(* Logix 5000 project; controller Safety vendor 1 type 14 code 86 rev 19.11; software revision 19.01; part 6 of 17 *)
(* tags used below, declared in another part *)
   ChgMe : BOOL;
   ESTOP_x201PB040 : DCI_STOP;   // OS1 Line EStop Pushbutton
   ESTOP_x211PB040 : DCI_STOP;   // OS2 Line EStop Pushbutton
   ESTOP_x221PB040 : DCI_STOP;   // OS3 Line EStop Pushbutton
   ESTOP_x231PB040 : DCI_STOP;   // OS4N Line EStop Pushbutton
   ESTOP_x241PB040 : DCI_STOP;   // OS4S Line EStop Pushbutton
   ESTOP_x251PB040 : DCI_STOP;   // OS5 Line EStop Pushbutton
   ESTOP_x261PB040 : DCI_STOP;   // OS6 Line EStop Pushbutton
   ESTOP_x271PB040 : DCI_STOP;   // OS8 Line EStop Pushbutton
   ESTOP_x281PB040 : DCI_STOP;   // OS9 Line EStop Pushbutton
   ESTOP_x291PB040 : DCI_STOP;   // OS11 Line EStop Pushbutton
   ESTOP_x301PB040 : DCI_STOP;   // OS13 Line EStop Pushbutton
   ESTOP_x311PB040 : DCI_STOP;   // OS14 Line EStop Pushbutton
   ESTOP_x311PB130 : DCI_STOP;   // OS14 Shear Estop Pushbutton
   ESTOP_x321PB040 : DCI_STOP;   // OS15 Line EStop Pushbutton
   ESTOP_x331PB040 : DCI_STOP;   // OS16 Line EStop Pushbutton
   ESTOP_x480PB470 : DCI_STOP;   // DPD Line EStop Pushbutton
   ESTOP_x480PB550 : DCI_STOP;   // DPD (In Pit) Line EStop Pushbutton
   ESTOP_x519LS470 : DCI_STOP;   // G1 Tripwire Line EStop
   ESTOP_x533PB470 : DCI_STOP;   // H1 Line EStop Pushbutton
   FUTURE : ALIAS FOR Diag_Tmp.1;   // FUTURE
   HB_Citect : BOOL;   // Heartbeat Citect Reflect
   Line_TotalMode : BOOL;   // Line TOTAL Mode ( 1= Total Mode) (0 = Coil to Coil)
   LineSts : UDT_SysStatus;
   ShearSts : UDT_ShearStatus;
   ToCitect : DINT[64];   // (To Citect)
   ToCitect4 : DINT[64];   // (To Citect4)
   x406LCA047 : ALIAS FOR A1:21:I.Pt00Data;   // North/South Light Curtain Output A
   x406LCB052 : ALIAS FOR A1:21:I.Pt01Data;   // North/South Light Curtain Output B
   x480PB470a : ALIAS FOR DPD:15:I.Pt00Data;   // Emergency Stop Pushbutton
   x480PB470b : ALIAS FOR DPD:15:I.Pt01Data;   // Emergency Stop Pushbutton
   x480PB550a : ALIAS FOR DPD:15:I.Pt02Data;   // Emergency Stop Pushbutton (In Pit)
   x480PB550b : ALIAS FOR DPD:15:I.Pt03Data;   // Emergency Stop Pushbutton (In Pit)
   x519LS470 : ALIAS FOR G1:12:I.Pt00Data;   // Tripwire Emergency Stop Limit Switch
   x613CR460 : ALIAS FOR CHPLC:1:I.Pt00Data;   // Unwind Operator Side Main Contactor Safety Relay
   x613CR510 : ALIAS FOR CHPLC:1:I.Pt01Data;   // Unwind Operator Side Drive Enable Safety Relay
   x613CR550 : ALIAS FOR CHPLC:1:I.Pt02Data;   // Unwind Drive Side Main Contactor Safety Relay
   x613CR590 : ALIAS FOR CHPLC:1:I.Pt03Data;   // Unwind Drive Side Drive Enable Safety Relay
   x613CR630 : ALIAS FOR CHPLC:1:I.Pt04Data;   // #1 Entry Bridle Roll 2 Main Contactor Safety Relay
   x613CR670 : ALIAS FOR CHPLC:1:I.Pt05Data;   // #1 Entry Bridle Roll 2 Drive Enable Safety Relay
   x613CR710 : ALIAS FOR CHPLC:1:I.Pt06Data;   // #2 Entry Bridle Roll 3 Main Contactor Safety Relay
   x613CR750 : ALIAS FOR CHPLC:1:I.Pt07Data;   // #2 Entry Bridle Roll 3 Drive Enable Safety Relay
   x614CR040 : ALIAS FOR CHPLC:2:I.Pt00Data;   // #1 Exit Bridle Roll 6 Main Contactor Safety Relay
   x614CR090 : ALIAS FOR CHPLC:2:I.Pt01Data;   // #1 Exit Bridle Roll 6 Drive Enable Safety Relay
   x614CR130 : ALIAS FOR CHPLC:2:I.Pt02Data;   // #2 Exit Bridle Roll 7 Main Contactor Safety Relay
   x614CR170 : ALIAS FOR CHPLC:2:I.Pt03Data;   // #2 Exit Bridle Roll 7 Drive Enable Safety Relay
   x614CR210 : ALIAS FOR CHPLC:2:I.Pt04Data;   // Rewind Main Contactor Safety Relay
   x614CR250 : ALIAS FOR CHPLC:2:I.Pt05Data;   // Rewind Drive Enable Safety Relay
   y406CR050 : ALIAS FOR A1:20:O.Pt00Data;   // Line Solenoid Safe Off
   y406CR090 : ALIAS FOR A1:20:O.Pt01Data;   // Coil Car Solenoid Safe Off
   y406CR120 : ALIAS FOR A1:20:O.Pt02Data;   // Spare
   y406CR170 : ALIAS FOR A1:20:O.Pt03Data;   // Spare
   y435CR050 : ALIAS FOR C1:12:O.Pt00Data;   // Solenoid Safe Off
   y451CR050 : ALIAS FOR D1:12:O.Pt00Data;   // Soleniod Safe Off
   y464CR050 : ALIAS FOR E1:10:O.Pt00Data;   // Soleniod Safe Off
   y480CR050 : ALIAS FOR DPD:14:O.Pt00Data;   // Solenoid Safe Off
   y507CR050 : ALIAS FOR F1:19:O.Pt00Data;   // Line Solenoid Safe Off
   y507CR090 : ALIAS FOR F1:19:O.Pt01Data;   // Rewind Coil Car Solenoid Safe Off
   y519CR050 : ALIAS FOR G1:11:O.Pt00Data;   // Line Solenoid Safe Off
   y533CR050 : ALIAS FOR H1:5:O.Pt00Data;   // Line Solenoid Safe Off
   y613CR460 : ALIAS FOR CHPLC:4:O.Pt00Data;   // Unwind Operator Side Main Contactor Safety Relay
   y613CR510 : ALIAS FOR CHPLC:4:O.Pt01Data;   // Unwind Operator Side Drive Enable Safety Relay
   y613CR550 : ALIAS FOR CHPLC:4:O.Pt02Data;   // Unwind Drive Side Main Contactor Safety Relay
   y613CR590 : ALIAS FOR CHPLC:4:O.Pt03Data;   // Unwind Drive Side Drive Enable Safety Relay
   y613CR630 : ALIAS FOR CHPLC:4:O.Pt04Data;   // #1 Entry Bridle Roll 2 Main Contactor Safety Relay
   y613CR670 : ALIAS FOR CHPLC:4:O.Pt05Data;   // #1 Entry Bridle Roll 2 Drive Enable Safety Relay
   y613CR710 : ALIAS FOR CHPLC:4:O.Pt06Data;   // #2 Entry Bridle Roll 3 Main Contactor Safety Relay
   y613CR750 : ALIAS FOR CHPLC:4:O.Pt07Data;   // #2 Entry Bridle Roll 3 Drive Enable Safety Relay
   y614CR040 : ALIAS FOR CHPLC:5:O.Pt00Data;   // #1 Exit Bridle Roll 6 Main Contactor Safety Relay
   y614CR090 : ALIAS FOR CHPLC:5:O.Pt01Data;   // #1 Exit Bridle Roll 6 Drive Enable Safety Relay
   y614CR130 : ALIAS FOR CHPLC:5:O.Pt02Data;   // #2 Exit Bridle Roll 7 Main Contactor Safety Relay
   y614CR170 : ALIAS FOR CHPLC:5:O.Pt03Data;   // #2 Exit Bridle Roll 7 Drive Enable Safety Relay
   y614CR210 : ALIAS FOR CHPLC:5:O.Pt04Data;   // Rewind Main Contactor Safety Relay
   y614CR250 : ALIAS FOR CHPLC:5:O.Pt05Data;   // Rewind Drive Enable Safety Relay
(* Comms, continued *)

ROUTINE ToCitect   (* ladder *)
// Safety Signals
// to Citect System
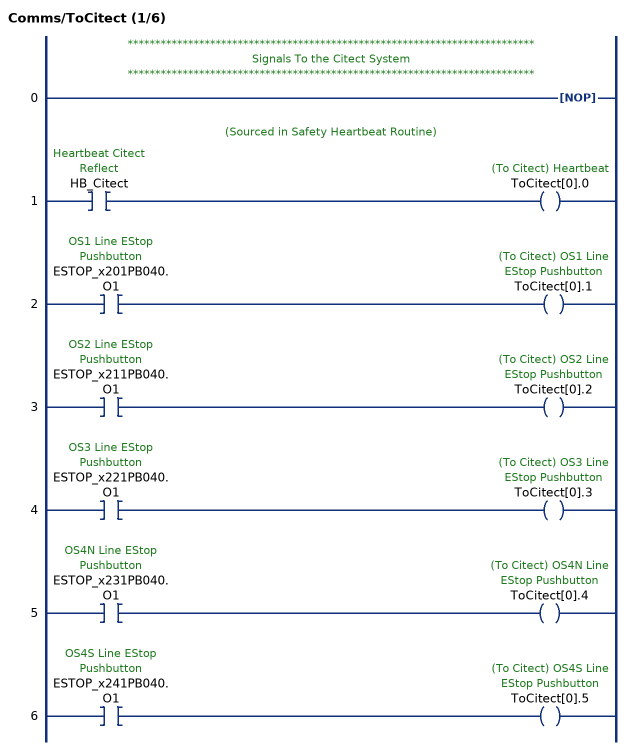
   // **************************************************************************
   // Signals To the Citect System
   // **************************************************************************
   0: NOP();
   // (Sourced in Safety Heartbeat Routine)
   1: XIC(HB_Citect)OTE(ToCitect[0].0);
   2: XIC(ESTOP_x201PB040.O1)OTE(ToCitect[0].1);
   3: XIC(ESTOP_x211PB040.O1)OTE(ToCitect[0].2);
   4: XIC(ESTOP_x221PB040.O1)OTE(ToCitect[0].3);
   5: XIC(ESTOP_x231PB040.O1)OTE(ToCitect[0].4);
   6: XIC(ESTOP_x241PB040.O1)OTE(ToCitect[0].5);
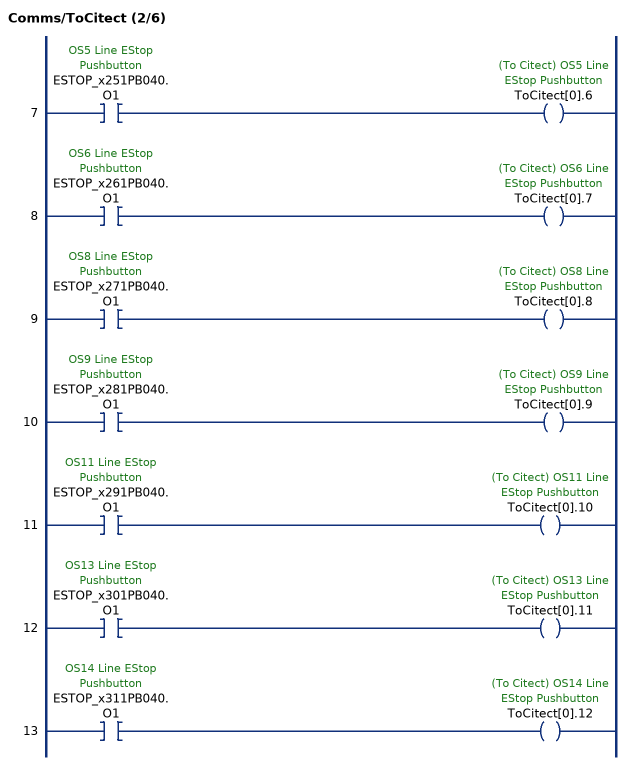
   7: XIC(ESTOP_x251PB040.O1)OTE(ToCitect[0].6);
   8: XIC(ESTOP_x261PB040.O1)OTE(ToCitect[0].7);
   9: XIC(ESTOP_x271PB040.O1)OTE(ToCitect[0].8);
   10: XIC(ESTOP_x281PB040.O1)OTE(ToCitect[0].9);
   11: XIC(ESTOP_x291PB040.O1)OTE(ToCitect[0].10);
   12: XIC(ESTOP_x301PB040.O1)OTE(ToCitect[0].11);
   13: XIC(ESTOP_x311PB040.O1)OTE(ToCitect[0].12);
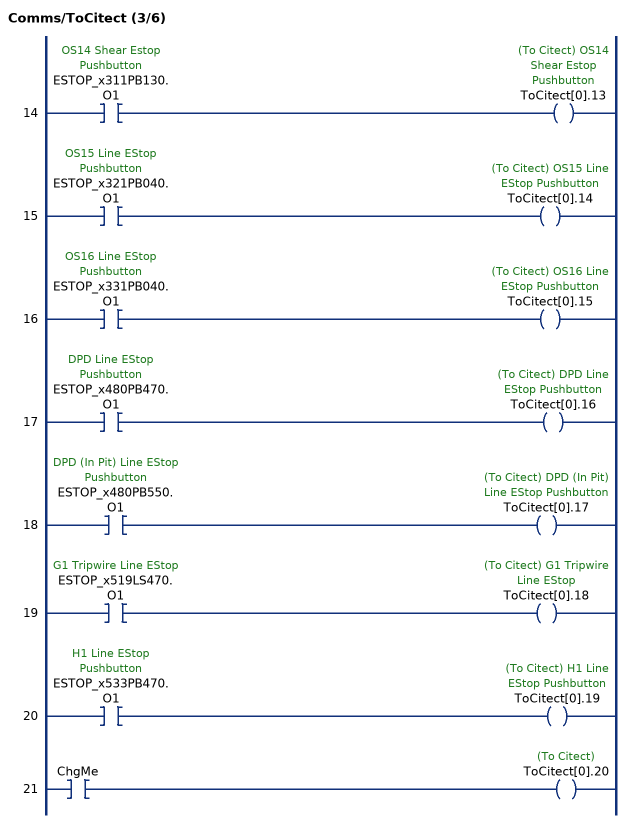
   14: XIC(ESTOP_x311PB130.O1)OTE(ToCitect[0].13);
   15: XIC(ESTOP_x321PB040.O1)OTE(ToCitect[0].14);
   16: XIC(ESTOP_x331PB040.O1)OTE(ToCitect[0].15);
   17: XIC(ESTOP_x480PB470.O1)OTE(ToCitect[0].16);
   18: XIC(ESTOP_x480PB550.O1)OTE(ToCitect[0].17);
   19: XIC(ESTOP_x519LS470.O1)OTE(ToCitect[0].18);
   20: XIC(ESTOP_x533PB470.O1)OTE(ToCitect[0].19);
   21: XIC(ChgMe)OTE(ToCitect[0].20);
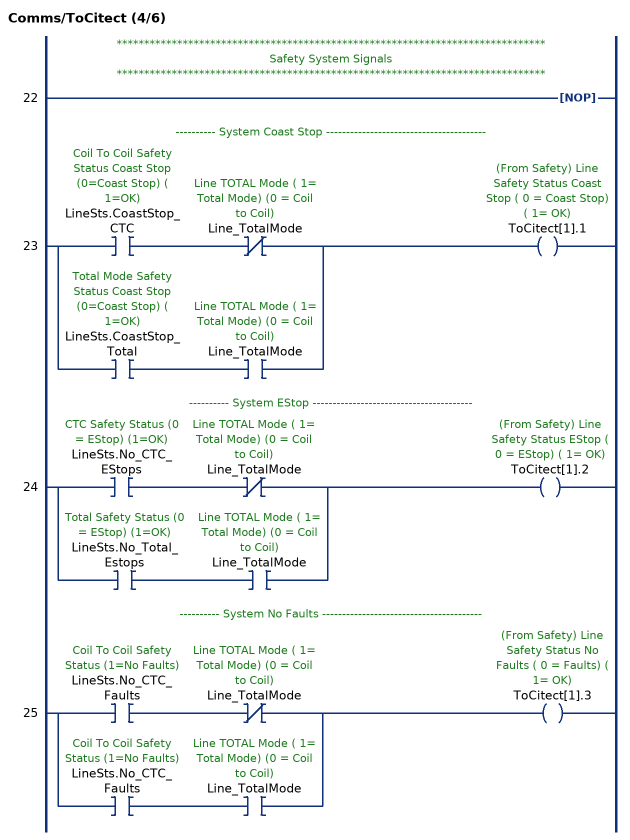
   // ******************************************************************************
   // Safety System Signals
   // ******************************************************************************
   22: NOP();
   // ---------- System Coast Stop ----------------------------------------
   23: [XIC(LineSts.CoastStop_CTC) XIO(Line_TotalMode) ,XIC(LineSts.CoastStop_Total) XIC(Line_TotalMode) ]OTE(ToCitect[1].1);
   // ---------- System EStop ----------------------------------------
   24: [XIC(LineSts.No_CTC_EStops) XIO(Line_TotalMode) ,XIC(LineSts.No_Total_Estops) XIC(Line_TotalMode) ]OTE(ToCitect[1].2);
   // ---------- System No Faults ----------------------------------------
   25: [XIC(LineSts.No_CTC_Faults) XIO(Line_TotalMode) ,XIC(LineSts.No_CTC_Faults) XIC(Line_TotalMode) ]OTE(ToCitect[1].3);
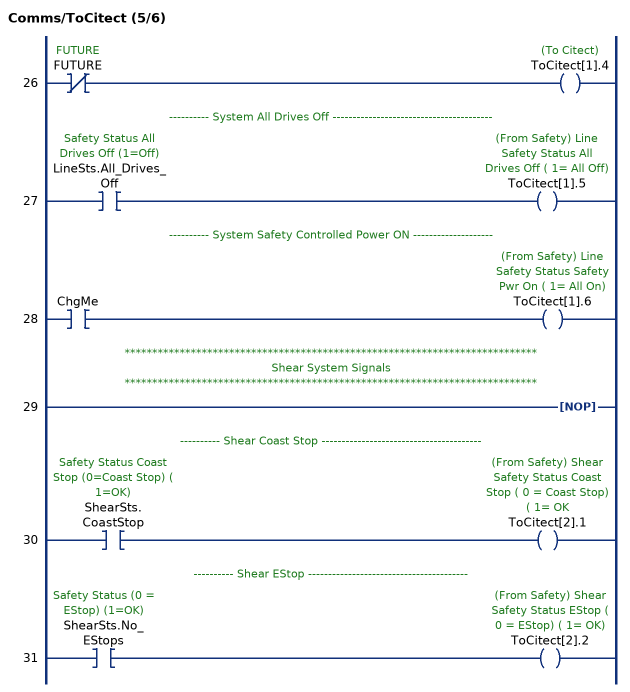
   26: XIO(FUTURE)OTE(ToCitect[1].4);
   // ---------- System All Drives Off ----------------------------------------
   27: XIC(LineSts.All_Drives_Off)OTE(ToCitect[1].5);
   // ---------- System Safety Controlled Power ON --------------------
   28: XIC(ChgMe)OTE(ToCitect[1].6);
   // ***************************************************************************
   // Shear System Signals
   // ***************************************************************************
   29: NOP();
   // ---------- Shear Coast Stop ----------------------------------------
   30: XIC(ShearSts.CoastStop)OTE(ToCitect[2].1);
   // ---------- Shear EStop ----------------------------------------
   31: XIC(ShearSts.No_EStops)OTE(ToCitect[2].2);
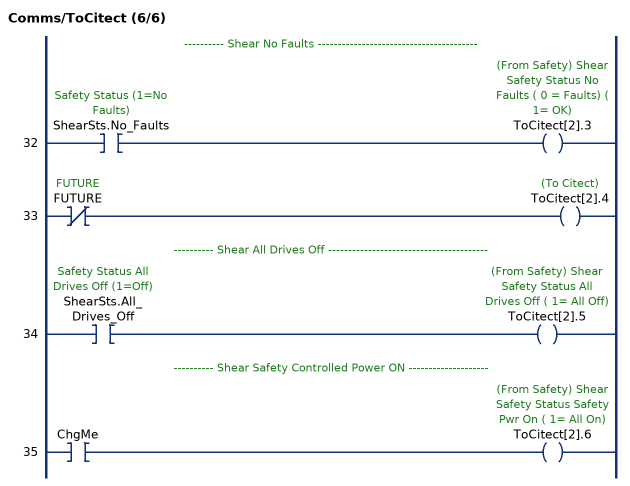
   // ---------- Shear No Faults ----------------------------------------
   32: XIC(ShearSts.No_Faults)OTE(ToCitect[2].3);
   33: XIO(FUTURE)OTE(ToCitect[2].4);
   // ---------- Shear All Drives Off ----------------------------------------
   34: XIC(ShearSts.All_Drives_Off)OTE(ToCitect[2].5);
   // ---------- Shear Safety Controlled Power ON --------------------
   35: XIC(ChgMe)OTE(ToCitect[2].6);
END_ROUTINE

ROUTINE ToCitect4   (* ladder *)
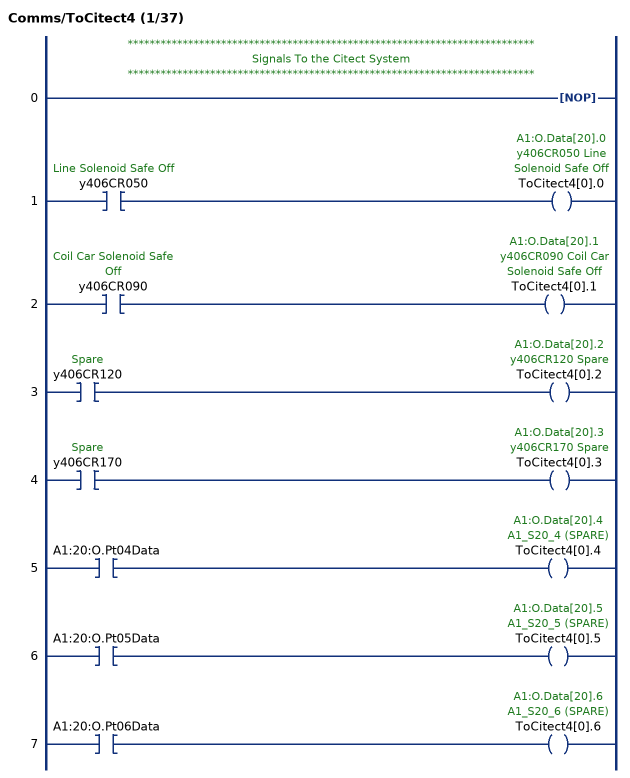
   // **************************************************************************
   // Signals To the Citect System
   // **************************************************************************
   0: NOP();
   1: XIC(y406CR050)OTE(ToCitect4[0].0);
   2: XIC(y406CR090)OTE(ToCitect4[0].1);
   3: XIC(y406CR120)OTE(ToCitect4[0].2);
   4: XIC(y406CR170)OTE(ToCitect4[0].3);
   5: XIC(A1:20:O.Pt04Data)OTE(ToCitect4[0].4);
   6: XIC(A1:20:O.Pt05Data)OTE(ToCitect4[0].5);
   7: XIC(A1:20:O.Pt06Data)OTE(ToCitect4[0].6);
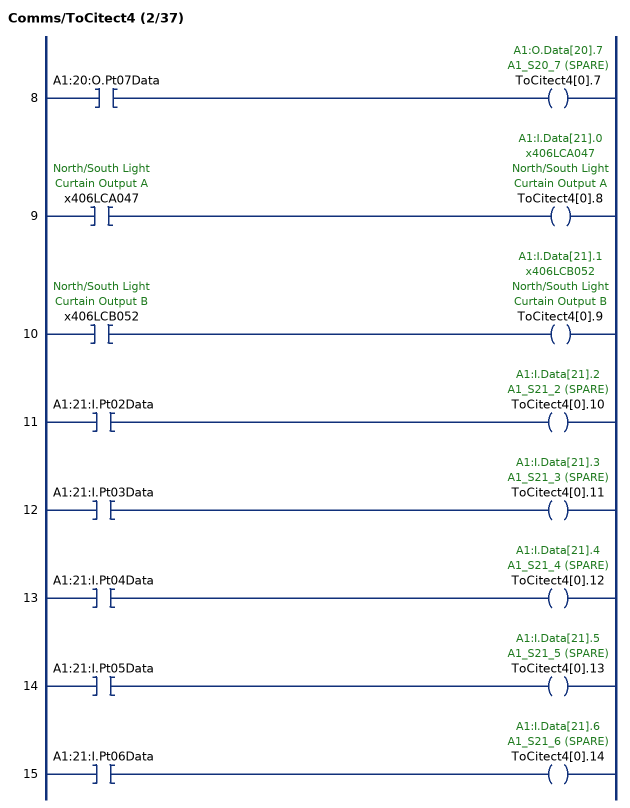
   8: XIC(A1:20:O.Pt07Data)OTE(ToCitect4[0].7);
   9: XIC(x406LCA047)OTE(ToCitect4[0].8);
   10: XIC(x406LCB052)OTE(ToCitect4[0].9);
   11: XIC(A1:21:I.Pt02Data)OTE(ToCitect4[0].10);
   12: XIC(A1:21:I.Pt03Data)OTE(ToCitect4[0].11);
   13: XIC(A1:21:I.Pt04Data)OTE(ToCitect4[0].12);
   14: XIC(A1:21:I.Pt05Data)OTE(ToCitect4[0].13);
   15: XIC(A1:21:I.Pt06Data)OTE(ToCitect4[0].14);
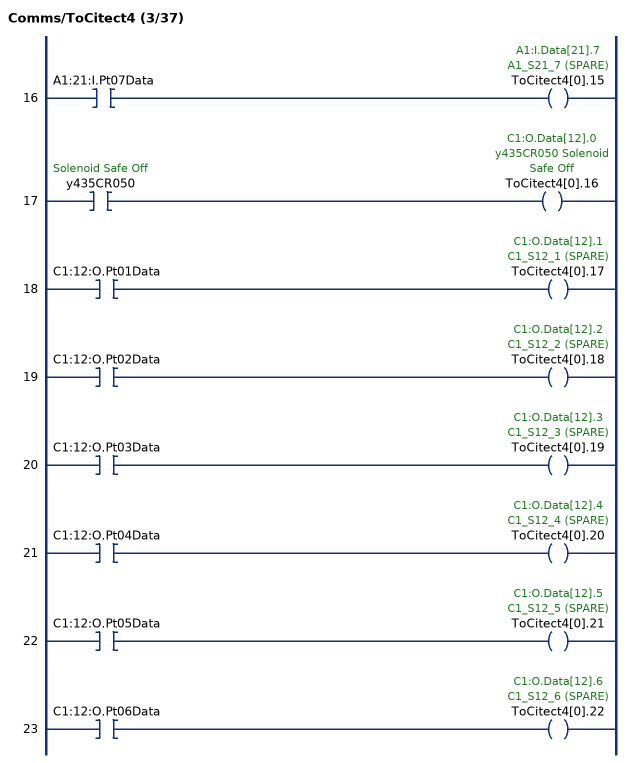
   16: XIC(A1:21:I.Pt07Data)OTE(ToCitect4[0].15);
   17: XIC(y435CR050)OTE(ToCitect4[0].16);
   18: XIC(C1:12:O.Pt01Data)OTE(ToCitect4[0].17);
   19: XIC(C1:12:O.Pt02Data)OTE(ToCitect4[0].18);
   20: XIC(C1:12:O.Pt03Data)OTE(ToCitect4[0].19);
   21: XIC(C1:12:O.Pt04Data)OTE(ToCitect4[0].20);
   22: XIC(C1:12:O.Pt05Data)OTE(ToCitect4[0].21);
   23: XIC(C1:12:O.Pt06Data)OTE(ToCitect4[0].22);
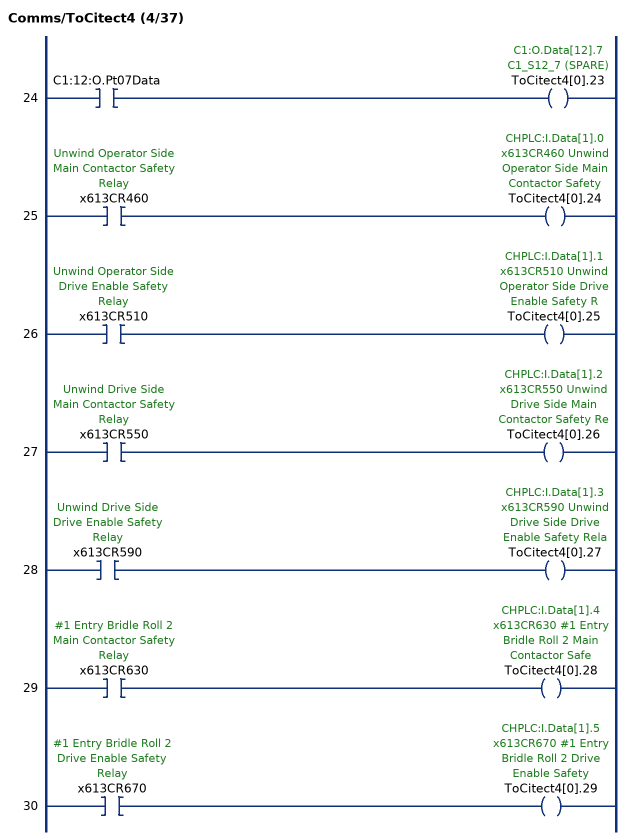
   24: XIC(C1:12:O.Pt07Data)OTE(ToCitect4[0].23);
   25: XIC(x613CR460)OTE(ToCitect4[0].24);
   26: XIC(x613CR510)OTE(ToCitect4[0].25);
   27: XIC(x613CR550)OTE(ToCitect4[0].26);
   28: XIC(x613CR590)OTE(ToCitect4[0].27);
   29: XIC(x613CR630)OTE(ToCitect4[0].28);
   30: XIC(x613CR670)OTE(ToCitect4[0].29);
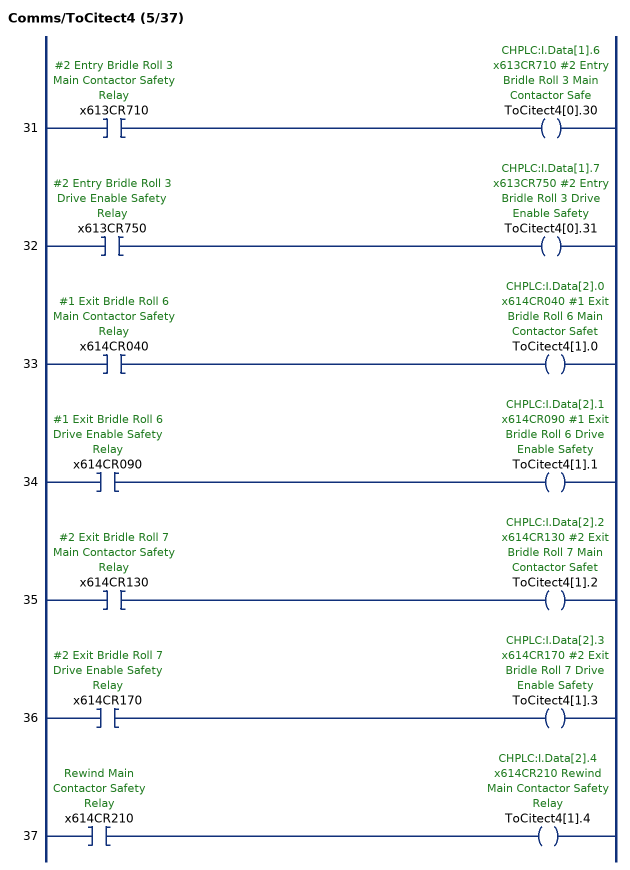
   31: XIC(x613CR710)OTE(ToCitect4[0].30);
   32: XIC(x613CR750)OTE(ToCitect4[0].31);
   33: XIC(x614CR040)OTE(ToCitect4[1].0);
   34: XIC(x614CR090)OTE(ToCitect4[1].1);
   35: XIC(x614CR130)OTE(ToCitect4[1].2);
   36: XIC(x614CR170)OTE(ToCitect4[1].3);
   37: XIC(x614CR210)OTE(ToCitect4[1].4);
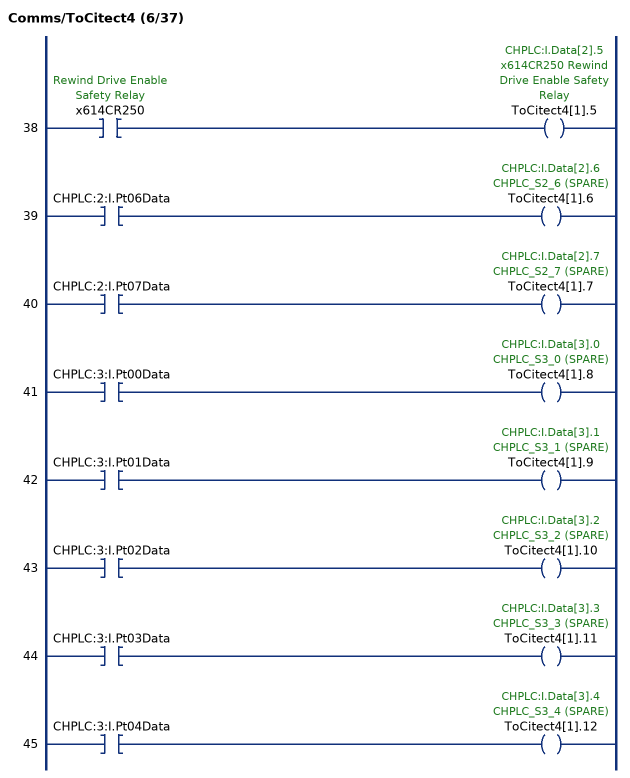
   38: XIC(x614CR250)OTE(ToCitect4[1].5);
   39: XIC(CHPLC:2:I.Pt06Data)OTE(ToCitect4[1].6);
   40: XIC(CHPLC:2:I.Pt07Data)OTE(ToCitect4[1].7);
   41: XIC(CHPLC:3:I.Pt00Data)OTE(ToCitect4[1].8);
   42: XIC(CHPLC:3:I.Pt01Data)OTE(ToCitect4[1].9);
   43: XIC(CHPLC:3:I.Pt02Data)OTE(ToCitect4[1].10);
   44: XIC(CHPLC:3:I.Pt03Data)OTE(ToCitect4[1].11);
   45: XIC(CHPLC:3:I.Pt04Data)OTE(ToCitect4[1].12);
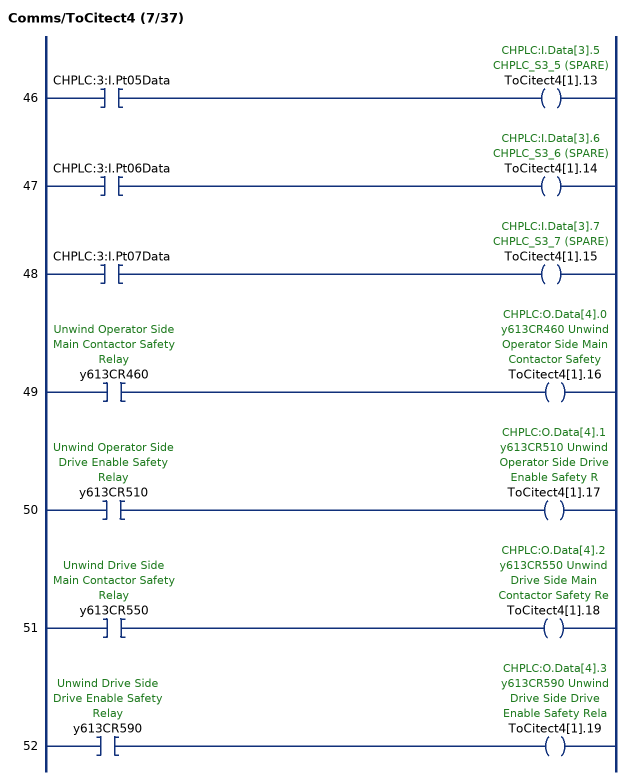
   46: XIC(CHPLC:3:I.Pt05Data)OTE(ToCitect4[1].13);
   47: XIC(CHPLC:3:I.Pt06Data)OTE(ToCitect4[1].14);
   48: XIC(CHPLC:3:I.Pt07Data)OTE(ToCitect4[1].15);
   49: XIC(y613CR460)OTE(ToCitect4[1].16);
   50: XIC(y613CR510)OTE(ToCitect4[1].17);
   51: XIC(y613CR550)OTE(ToCitect4[1].18);
   52: XIC(y613CR590)OTE(ToCitect4[1].19);
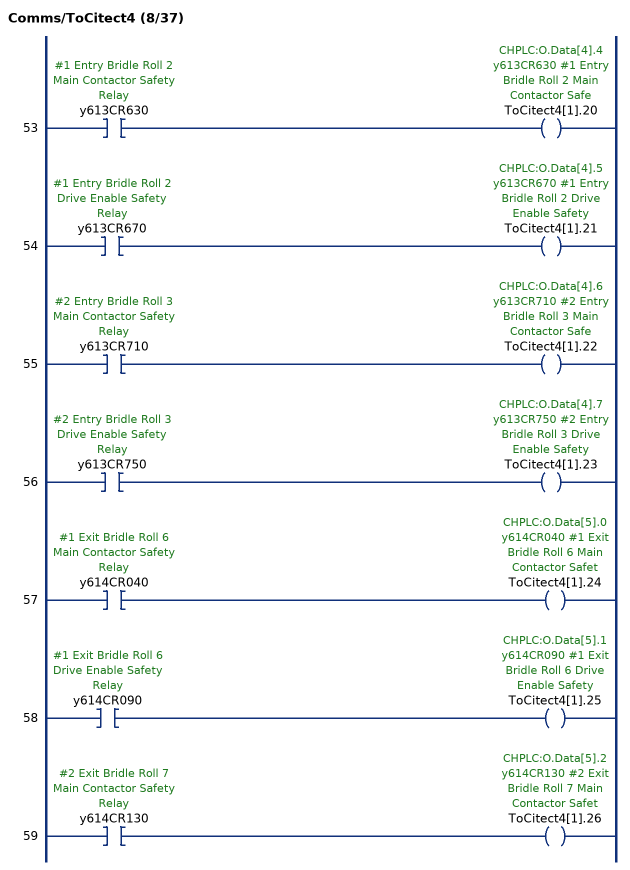
   53: XIC(y613CR630)OTE(ToCitect4[1].20);
   54: XIC(y613CR670)OTE(ToCitect4[1].21);
   55: XIC(y613CR710)OTE(ToCitect4[1].22);
   56: XIC(y613CR750)OTE(ToCitect4[1].23);
   57: XIC(y614CR040)OTE(ToCitect4[1].24);
   58: XIC(y614CR090)OTE(ToCitect4[1].25);
   59: XIC(y614CR130)OTE(ToCitect4[1].26);
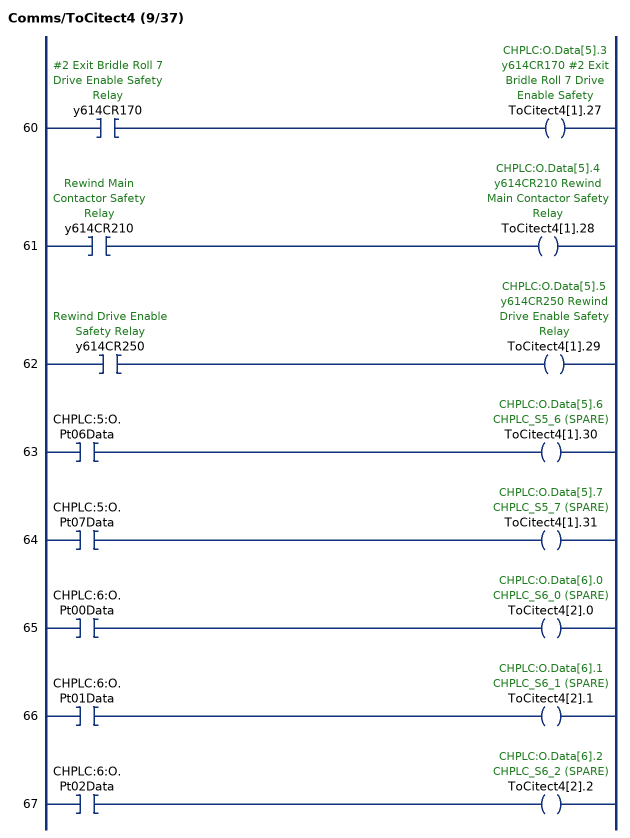
   60: XIC(y614CR170)OTE(ToCitect4[1].27);
   61: XIC(y614CR210)OTE(ToCitect4[1].28);
   62: XIC(y614CR250)OTE(ToCitect4[1].29);
   63: XIC(CHPLC:5:O.Pt06Data)OTE(ToCitect4[1].30);
   64: XIC(CHPLC:5:O.Pt07Data)OTE(ToCitect4[1].31);
   65: XIC(CHPLC:6:O.Pt00Data)OTE(ToCitect4[2].0);
   66: XIC(CHPLC:6:O.Pt01Data)OTE(ToCitect4[2].1);
   67: XIC(CHPLC:6:O.Pt02Data)OTE(ToCitect4[2].2);
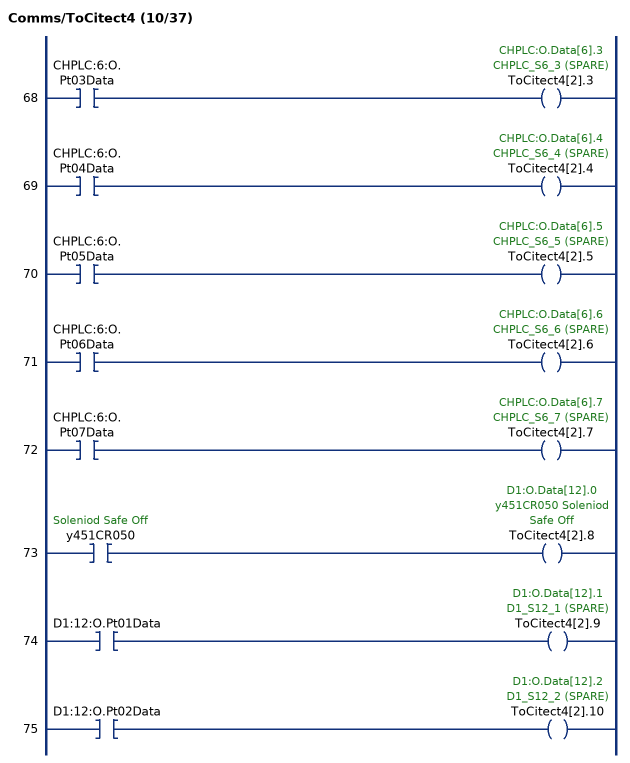
   68: XIC(CHPLC:6:O.Pt03Data)OTE(ToCitect4[2].3);
   69: XIC(CHPLC:6:O.Pt04Data)OTE(ToCitect4[2].4);
   70: XIC(CHPLC:6:O.Pt05Data)OTE(ToCitect4[2].5);
   71: XIC(CHPLC:6:O.Pt06Data)OTE(ToCitect4[2].6);
   72: XIC(CHPLC:6:O.Pt07Data)OTE(ToCitect4[2].7);
   73: XIC(y451CR050)OTE(ToCitect4[2].8);
   74: XIC(D1:12:O.Pt01Data)OTE(ToCitect4[2].9);
   75: XIC(D1:12:O.Pt02Data)OTE(ToCitect4[2].10);
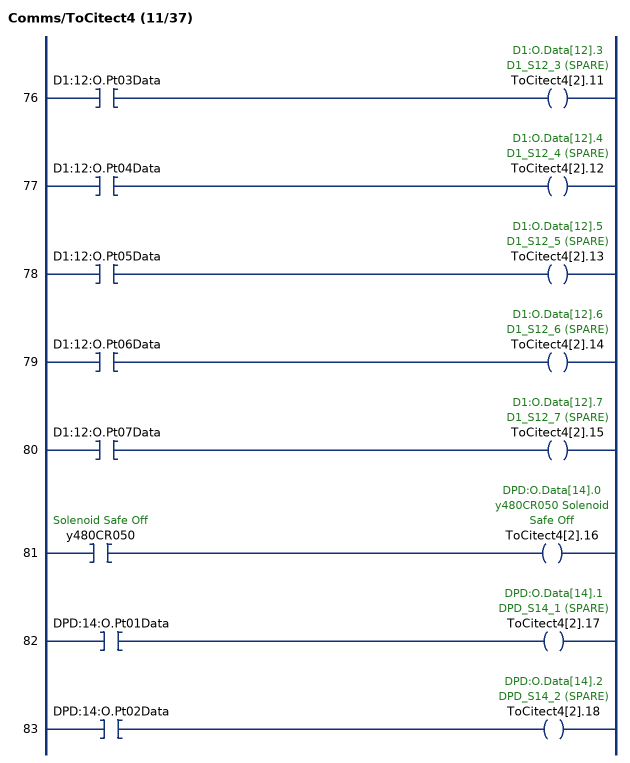
   76: XIC(D1:12:O.Pt03Data)OTE(ToCitect4[2].11);
   77: XIC(D1:12:O.Pt04Data)OTE(ToCitect4[2].12);
   78: XIC(D1:12:O.Pt05Data)OTE(ToCitect4[2].13);
   79: XIC(D1:12:O.Pt06Data)OTE(ToCitect4[2].14);
   80: XIC(D1:12:O.Pt07Data)OTE(ToCitect4[2].15);
   81: XIC(y480CR050)OTE(ToCitect4[2].16);
   82: XIC(DPD:14:O.Pt01Data)OTE(ToCitect4[2].17);
   83: XIC(DPD:14:O.Pt02Data)OTE(ToCitect4[2].18);
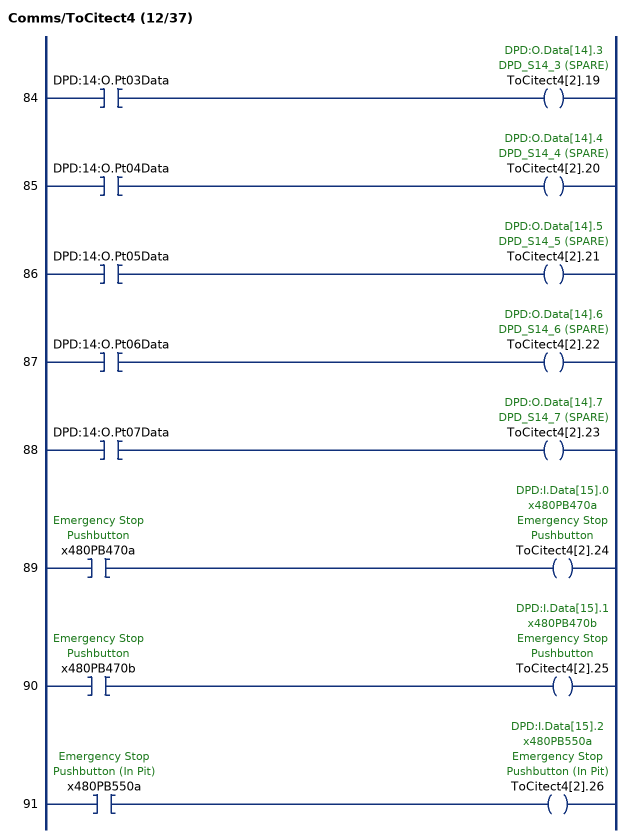
   84: XIC(DPD:14:O.Pt03Data)OTE(ToCitect4[2].19);
   85: XIC(DPD:14:O.Pt04Data)OTE(ToCitect4[2].20);
   86: XIC(DPD:14:O.Pt05Data)OTE(ToCitect4[2].21);
   87: XIC(DPD:14:O.Pt06Data)OTE(ToCitect4[2].22);
   88: XIC(DPD:14:O.Pt07Data)OTE(ToCitect4[2].23);
   89: XIC(x480PB470a)OTE(ToCitect4[2].24);
   90: XIC(x480PB470b)OTE(ToCitect4[2].25);
   91: XIC(x480PB550a)OTE(ToCitect4[2].26);
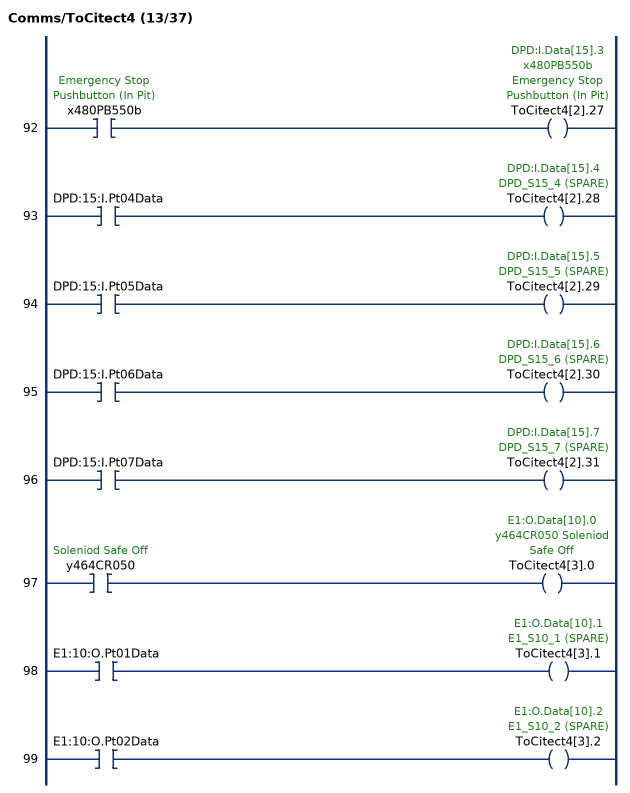
   92: XIC(x480PB550b)OTE(ToCitect4[2].27);
   93: XIC(DPD:15:I.Pt04Data)OTE(ToCitect4[2].28);
   94: XIC(DPD:15:I.Pt05Data)OTE(ToCitect4[2].29);
   95: XIC(DPD:15:I.Pt06Data)OTE(ToCitect4[2].30);
   96: XIC(DPD:15:I.Pt07Data)OTE(ToCitect4[2].31);
   97: XIC(y464CR050)OTE(ToCitect4[3].0);
   98: XIC(E1:10:O.Pt01Data)OTE(ToCitect4[3].1);
   99: XIC(E1:10:O.Pt02Data)OTE(ToCitect4[3].2);
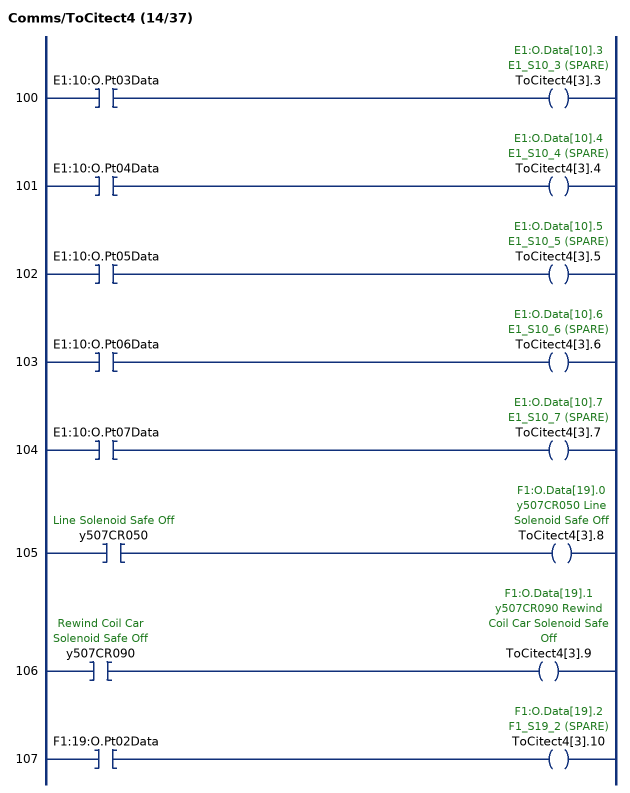
   100: XIC(E1:10:O.Pt03Data)OTE(ToCitect4[3].3);
   101: XIC(E1:10:O.Pt04Data)OTE(ToCitect4[3].4);
   102: XIC(E1:10:O.Pt05Data)OTE(ToCitect4[3].5);
   103: XIC(E1:10:O.Pt06Data)OTE(ToCitect4[3].6);
   104: XIC(E1:10:O.Pt07Data)OTE(ToCitect4[3].7);
   105: XIC(y507CR050)OTE(ToCitect4[3].8);
   106: XIC(y507CR090)OTE(ToCitect4[3].9);
   107: XIC(F1:19:O.Pt02Data)OTE(ToCitect4[3].10);
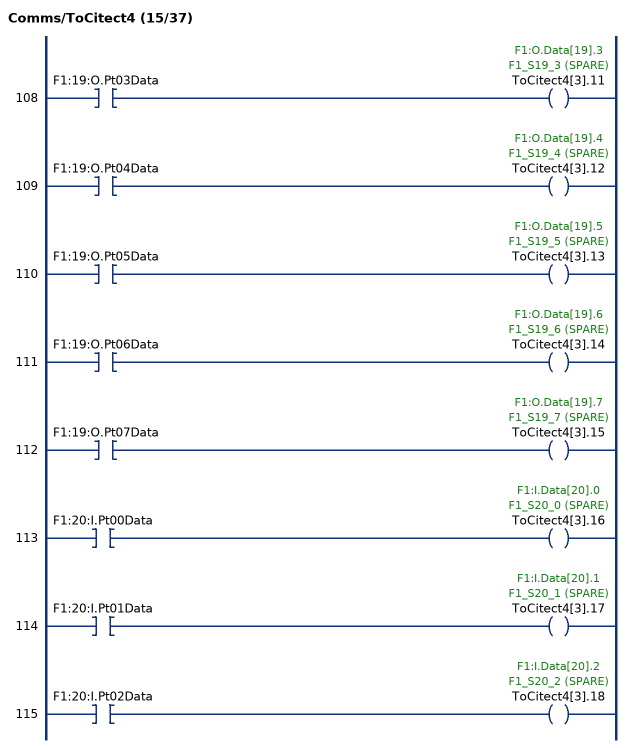
   108: XIC(F1:19:O.Pt03Data)OTE(ToCitect4[3].11);
   109: XIC(F1:19:O.Pt04Data)OTE(ToCitect4[3].12);
   110: XIC(F1:19:O.Pt05Data)OTE(ToCitect4[3].13);
   111: XIC(F1:19:O.Pt06Data)OTE(ToCitect4[3].14);
   112: XIC(F1:19:O.Pt07Data)OTE(ToCitect4[3].15);
   113: XIC(F1:20:I.Pt00Data)OTE(ToCitect4[3].16);
   114: XIC(F1:20:I.Pt01Data)OTE(ToCitect4[3].17);
   115: XIC(F1:20:I.Pt02Data)OTE(ToCitect4[3].18);
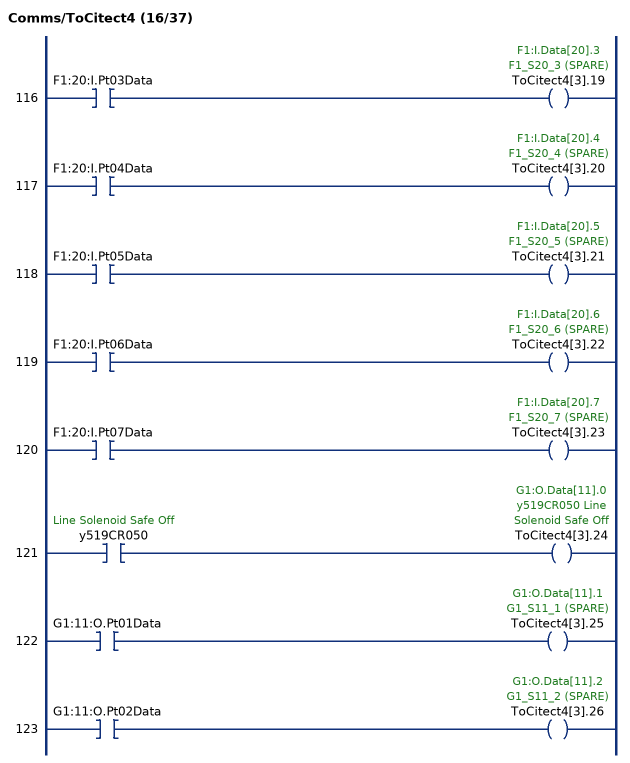
   116: XIC(F1:20:I.Pt03Data)OTE(ToCitect4[3].19);
   117: XIC(F1:20:I.Pt04Data)OTE(ToCitect4[3].20);
   118: XIC(F1:20:I.Pt05Data)OTE(ToCitect4[3].21);
   119: XIC(F1:20:I.Pt06Data)OTE(ToCitect4[3].22);
   120: XIC(F1:20:I.Pt07Data)OTE(ToCitect4[3].23);
   121: XIC(y519CR050)OTE(ToCitect4[3].24);
   122: XIC(G1:11:O.Pt01Data)OTE(ToCitect4[3].25);
   123: XIC(G1:11:O.Pt02Data)OTE(ToCitect4[3].26);
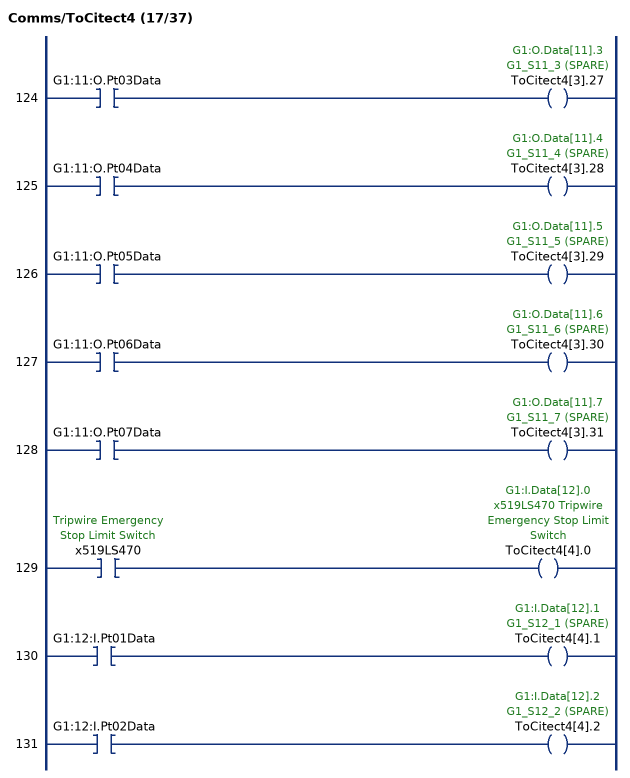
   124: XIC(G1:11:O.Pt03Data)OTE(ToCitect4[3].27);
   125: XIC(G1:11:O.Pt04Data)OTE(ToCitect4[3].28);
   126: XIC(G1:11:O.Pt05Data)OTE(ToCitect4[3].29);
   127: XIC(G1:11:O.Pt06Data)OTE(ToCitect4[3].30);
   128: XIC(G1:11:O.Pt07Data)OTE(ToCitect4[3].31);
   129: XIC(x519LS470)OTE(ToCitect4[4].0);
   130: XIC(G1:12:I.Pt01Data)OTE(ToCitect4[4].1);
   131: XIC(G1:12:I.Pt02Data)OTE(ToCitect4[4].2);
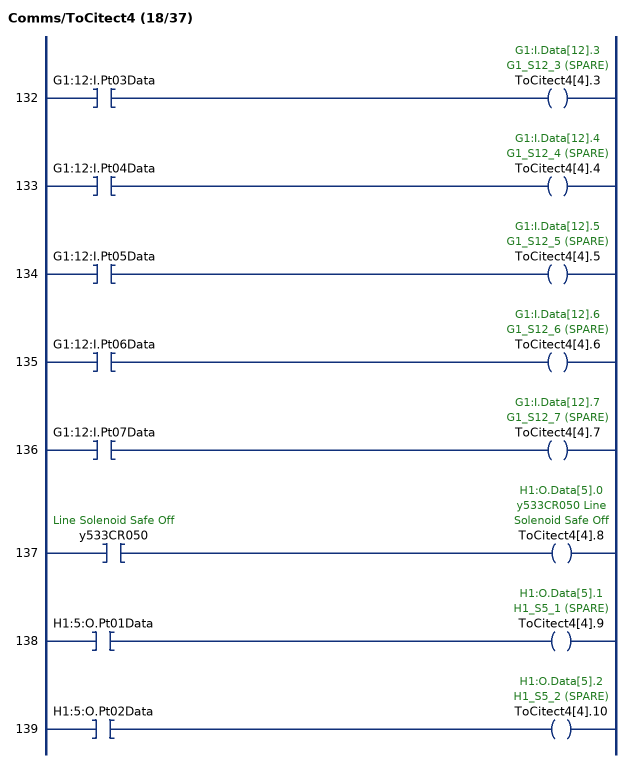
   132: XIC(G1:12:I.Pt03Data)OTE(ToCitect4[4].3);
   133: XIC(G1:12:I.Pt04Data)OTE(ToCitect4[4].4);
   134: XIC(G1:12:I.Pt05Data)OTE(ToCitect4[4].5);
   135: XIC(G1:12:I.Pt06Data)OTE(ToCitect4[4].6);
   136: XIC(G1:12:I.Pt07Data)OTE(ToCitect4[4].7);
   137: XIC(y533CR050)OTE(ToCitect4[4].8);
   138: XIC(H1:5:O.Pt01Data)OTE(ToCitect4[4].9);
   139: XIC(H1:5:O.Pt02Data)OTE(ToCitect4[4].10);
